Fanuc TP program (LS listing): UP023.LS

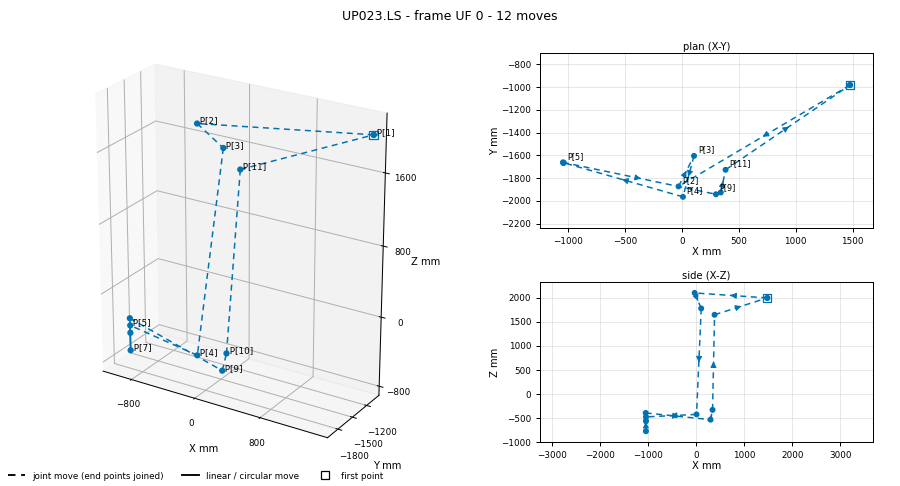
[picture p0: tool path of UP023.LS in frame UF 0, 12 of 12 moves have a stored position in this frame; points joined in program order, loops and branches not executed]
/PROG  UP023
/ATTR
OWNER		= GME;
COMMENT		= "Dejar en ST1620";
PROG_SIZE	= 5438;
CREATE		= DATE 96-03-29  TIME 13:09:40;
MODIFIED	= DATE 23-07-01  TIME 02:04:06;
FILE_NAME	= UP023;
VERSION		= 0;
LINE_COUNT	= 23;
MEMORY_SIZE	= 10066;
PROTECT		= READ_WRITE;
TCD:  STACK_SIZE	= 500,
      TASK_PRIORITY	= 50,
      TIME_SLICE	= 0,
      BUSY_LAMP_OFF	= 0,
      ABORT_REQUEST	= 0,
      PAUSE_REQUEST	= 0;
DEFAULT_GROUP	= 1,1,1,1,*;
CONTROL_CODE	= 00000000 00000000;
/APPL
/MN
   1:  UFRAME_NUM=0 ;
   2:  UTOOL_NUM=1 ;
   3:  PAYLOAD[2] ;
   4:  !Apagar Perfil Lib. 76 vs ST1620 ;
   5:  !Encender Anticol. 1 vs 1630R01 ;
   6:J P[1] 100% CNT0 ACC100 TB    .10sec,P-SPS    ;
      1:  TC_ONLINE (ON) ;
      2:  DO[23]=OFF ;
      3:  TIMER[5]=RESET ;
      4:  TIMER[5]=START ;
      5:  CALL MAKRO050    ;
      6:  !Lib. de Herramientas ;
      7:  DO[80]=ON ;
      8:  DO[79]=ON ;
      9:  DO[78]=OFF ;
     10:  DO[77]=OFF ;
     11:  DO[76]=ON ;
     12:  DO[74]=OFF ;
     13:  !Lib. de Anticolisiones ;
     14:  DO[41]=ON ;
     15:  DO[42]=ON ;
     16:  DO[43]=ON ;
     17:  DO[44]=ON ;
     18:  DO[47]=ON ;
     19:  DO[48]=ON ;
     20:  !Apagar Pos. Base ;
     21:  DO[15]=OFF ;
     22:  !Robot en Trayectoria ;
     23:  DO[16]=ON ;
     24:  WAIT (DI[76] AND !DI[62] AND DI[61] AND M[31] AND M[34])    ;
     25:  DO[76]=OFF ;
     26:  !Encender Anticolisiones ;
     27:  DO[81]=ON ;
     28:  CALL MAKRO020    ;
     29:  WAIT (DI[23])    ;
     30:  DO[23]=ON ;
     31:  TC_ONLINE (DI[41] AND !DI[62] AND DI[61] AND DI[76] AND M[1] AND M[30] AND M[31] AND M[34] AND M[95] AND M[96]) ;
       ------ ;
   7:J P[2] 100% CNT100 ACC100 TB   0.00sec,P-SPS    ;
      1:  TC_ONLINE (DI[41] AND !DI[62] AND DI[61] AND DI[76] AND M[1] AND M[30] AND M[31] AND M[34] AND M[95] AND M[96]) ;
       ------ ;
   8:J P[3] 100% CNT100 ACC100 TB   0.00sec,P-SPS    ;
      1:  TC_ONLINE (DI[41] AND !DI[62] AND DI[61] AND DI[76] AND M[1] AND M[30] AND M[31] AND M[34] AND M[95] AND M[96]) ;
       ------ ;
   9:J P[4] 100% CNT100 ACC100 TB   0.00sec,P-SPS    ;
      1:  TC_ONLINE (DI[41] AND !DI[62] AND DI[61] AND DI[76] AND M[1] AND M[30] AND M[31] AND M[34] AND M[95] AND M[96]) ;
       ------ ;
  10:J P[5] 100% CNT100 ACC100 TB   0.00sec,P-SPS    ;
      1:  TC_ONLINE (DI[41] AND !DI[62] AND DI[61] AND DI[76] AND M[1] AND M[30] AND M[31] AND M[34] AND M[95] AND M[96]) ;
       ------ ;
  11:J P[6] 100% CNT100 ACC100 TB   0.00sec,P-SPS    ;
      1:  TC_ONLINE (DI[41] AND DI[76] AND M[1] AND M[30] AND M[31] AND M[34] AND M[95] AND M[96]) ;
       ------ ;
  12:  !En Posicion ST1620 ;
  13:  !Dejar Pieza en ST1620 ;
  14:  !Fin de Trabajo 3 ;
  15:L P[7] 1500mm/sec CNT0 ACC100 TB    .10sec,P-SPS    ;
      1:  TC_ONLINE (ON) ;
      2:  DO[23]=OFF ;
      3:  WAIT ((DI[62] AND !DI[61]) OR DI[15])    ;
      4:  DO[74]=ON ;
      5:  CALL MAKRO003    ;
      6:  WAIT (DI[75])    ;
      7:  DO[74]=OFF ;
      8:  F[2]=(ON) ;
      9:  CALL MAKRO342    ;
     10:  CALL MAKRO340    ;
     11:  WAIT (M[33])    ;
     12:  WAIT (DI[23])    ;
     13:  DO[23]=ON ;
     14:  TC_ONLINE (DI[41] AND !DI[61] AND DI[62] AND DI[75] AND M[30] AND M[31] AND M[33] AND M[95] AND M[96]) ;
       ------ ;
  16:  PAYLOAD[1] ;
  17:L P[8] 2000mm/sec CNT100 ACC100 TB   0.00sec,P-SPS    ;
      1:  TC_ONLINE (DI[41] AND !DI[61] AND DI[62] AND DI[75] AND M[2] AND M[30] AND M[31] AND M[33] AND M[95] AND M[96]) ;
       ------ ;
  18:J P[9] 100% CNT100 ACC100 TB   0.00sec,P-SPS    ;
      1:  TC_ONLINE (DI[41] AND !DI[61] AND DI[62] AND DI[75] AND M[2] AND M[30] AND M[31] AND M[33] AND M[95] AND M[96]) ;
       ------ ;
  19:J P[10] 100% CNT100 ACC100 TB   0.00sec,P-SPS    ;
      1:  TC_ONLINE (ON) ;
      2:  DO[41]=ON ;
      3:  DO[76]=ON ;
      4:  TC_ONLINE (M[2] AND M[30] AND M[31] AND M[33] AND M[95] AND M[96]) ;
       ------ ;
  20:J P[11] 100% CNT100 ACC100 TB   0.00sec,P-SPS    ;
      1:  TC_ONLINE (M[2] AND M[30] AND M[31] AND M[33] AND M[95] AND M[96]) ;
       ------ ;
  21:  !Encender Perfil Lib 76 vs ST1620 ;
  22:  !Apagar Anticol. 1 vs 1630R01 ;
  23:J P[12] 100% CNT0 ACC100 TB    .10sec,P-SPS    ;
      1:  TC_ONLINE (ON) ;
      2:  DO[23]=OFF ;
      3:  TIMER[5]=STOP ;
      4:  WAIT (DI[23])    ;
      5:  DO[23]=ON ;
      6:  TC_ONLINE (M[2] AND M[30] AND M[31] AND M[33] AND M[95] AND M[96]) ;
       ------ ;
/POS
P[1]{
   GP1:
	UF : 0, UT : 1,		CONFIG : 'F U T, 0, 1, 0',
	X =  1478.134  mm,	Y =  -981.143  mm,	Z =  1998.395  mm,
	W =   145.269 deg,	P =    62.134 deg,	R =   -76.624 deg
   GP2:
	UF : 0, UT : 1,
	J1=   100.000  mm
   GP3:
	UF : 0, UT : 1,
	J1=     0.000  mm
   GP4:
	UF : 0, UT : 1,
	J1=     0.000  mm
};
P[2]{
   GP1:
	UF : 0, UT : 1,		CONFIG : 'F U T, 0, 0, 0',
	X =   -31.554  mm,	Y = -1873.422  mm,	Z =  2101.961  mm,
	W =    60.915 deg,	P =   -11.606 deg,	R =  -123.381 deg
   GP2:
	UF : 0, UT : 1,
	J1=   100.000  mm
   GP3:
	UF : 0, UT : 1,
	J1=     0.000  mm
   GP4:
	UF : 0, UT : 1,
	J1=     0.000  mm
};
P[3]{
   GP1:
	UF : 0, UT : 1,		CONFIG : 'F U T, 0, 0, 0',
	X =   104.894  mm,	Y = -1604.479  mm,	Z =  1780.030  mm,
	W =    42.682 deg,	P =     7.009 deg,	R =  -104.181 deg
   GP2:
	UF : 0, UT : 1,
	J1=   100.000  mm
   GP3:
	UF : 0, UT : 1,
	J1=     0.000  mm
   GP4:
	UF : 0, UT : 1,
	J1=     0.000  mm
};
P[4]{
   GP1:
	UF : 0, UT : 1,		CONFIG : 'F U T, 0, 0, 0',
	X =     7.472  mm,	Y = -1965.095  mm,	Z =  -422.745  mm,
	W =   161.299 deg,	P =    88.939 deg,	R =    13.610 deg
   GP2:
	UF : 0, UT : 1,
	J1=   100.000  mm
   GP3:
	UF : 0, UT : 1,
	J1=     0.000  mm
   GP4:
	UF : 0, UT : 1,
	J1=     0.000  mm
};
P[5]{
   GP1:
	UF : 0, UT : 1,		CONFIG : 'F U T, 0, 0, 0',
	X = -1043.496  mm,	Y = -1664.947  mm,	Z =  -474.897  mm,
	W =  -120.640 deg,	P =    84.826 deg,	R =    62.088 deg
   GP2:
	UF : 0, UT : 1,
	J1=   100.000  mm
   GP3:
	UF : 0, UT : 1,
	J1=     0.000  mm
   GP4:
	UF : 0, UT : 1,
	J1=     0.000  mm
};
P[6]{
   GP1:
	UF : 0, UT : 1,		CONFIG : 'F U T, 0, 0, 0',
	X = -1043.635  mm,	Y = -1664.947  mm,	Z =  -562.735  mm,
	W =   161.526 deg,	P =    88.942 deg,	R =   -18.404 deg
   GP2:
	UF : 0, UT : 1,
	J1=   100.000  mm
   GP3:
	UF : 0, UT : 1,
	J1=     0.000  mm
   GP4:
	UF : 0, UT : 1,
	J1=     0.000  mm
};
P[7]{
   GP1:
	UF : 0, UT : 1,		CONFIG : 'F U T, 0, 0, 0',
	X = -1044.280  mm,	Y = -1666.708  mm,	Z =  -771.997  mm,
	W =   165.038 deg,	P =    88.336 deg,	R =   -15.168 deg
   GP2:
	UF : 0, UT : 1,
	J1=   100.000  mm
   GP3:
	UF : 0, UT : 1,
	J1=     0.000  mm
   GP4:
	UF : 0, UT : 1,
	J1=     0.000  mm
};
P[8]{
   GP1:
	UF : 0, UT : 1,		CONFIG : 'F U T, 0, 0, 0',
	X = -1048.665  mm,	Y = -1662.047  mm,	Z =  -392.802  mm,
	W =   161.301 deg,	P =    88.939 deg,	R =   -18.842 deg
   GP2:
	UF : 0, UT : 1,
	J1=   100.000  mm
   GP3:
	UF : 0, UT : 1,
	J1=     0.000  mm
   GP4:
	UF : 0, UT : 1,
	J1=     0.000  mm
};
P[9]{
   GP1:
	UF : 0, UT : 1,		CONFIG : 'F U T, 0, 0, 0',
	X =   297.995  mm,	Y = -1942.514  mm,	Z =  -532.003  mm,
	W =   161.302 deg,	P =    88.939 deg,	R =    22.132 deg
   GP2:
	UF : 0, UT : 1,
	J1=   100.000  mm
   GP3:
	UF : 0, UT : 1,
	J1=     0.000  mm
   GP4:
	UF : 0, UT : 1,
	J1=     0.000  mm
};
P[10]{
   GP1:
	UF : 0, UT : 1,		CONFIG : 'F U T, 0, 0, 0',
	X =   340.526  mm,	Y = -1926.759  mm,	Z =  -328.520  mm,
	W =  -152.699 deg,	P =    88.950 deg,	R =    49.000 deg
   GP2:
	UF : 0, UT : 1,
	J1=   100.000  mm
   GP3:
	UF : 0, UT : 1,
	J1=     0.000  mm
   GP4:
	UF : 0, UT : 1,
	J1=     0.000  mm
};
P[11]{
   GP1:
	UF : 0, UT : 1,		CONFIG : 'F U T, 0, 0, 0',
	X =   382.420  mm,	Y = -1726.964  mm,	Z =  1648.257  mm,
	W =    51.669 deg,	P =    17.663 deg,	R =  -111.528 deg
   GP2:
	UF : 0, UT : 1,
	J1=   100.000  mm
   GP3:
	UF : 0, UT : 1,
	J1=     0.000  mm
   GP4:
	UF : 0, UT : 1,
	J1=     0.000  mm
};
P[12]{
   GP1:
	UF : 0, UT : 1,		CONFIG : 'F U T, 0, 1, 0',
	X =  1478.134  mm,	Y =  -981.144  mm,	Z =  1998.395  mm,
	W =   145.269 deg,	P =    62.134 deg,	R =   -76.624 deg
   GP2:
	UF : 0, UT : 1,
	J1=   100.000  mm
   GP3:
	UF : 0, UT : 1,
	J1=     0.000  mm
   GP4:
	UF : 0, UT : 1,
	J1=     0.000  mm
};
/END
